FUNCTION_BLOCK SPECIALSTRING_EQ (* Basic Function Block Type *)
  (* Standard: 61499-2 *)
  (* Version 0.0, 2015-11-04, 4DIAC-IDE, 4DIAC-Consortium *)
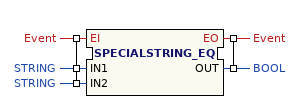
  EVENT_INPUT
    EI WITH IN1, IN2; (* Initialization Request *)
  END_EVENT
  EVENT_OUTPUT
    EO WITH OUT; (* Initialization Confirm *)
  END_EVENT
  VAR_INPUT
    IN1 : STRING;
    IN2 : STRING;
  END_VAR
  VAR_OUTPUT
    OUT : BOOL;
  END_VAR
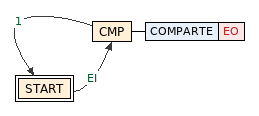
  EC_STATES
    START; (* Initial State *)
    CMP : COMPARTE -> EO; (* Initialization *)
  END_STATES
  EC_TRANSITIONS
    START TO CMP := EI;
    CMP TO START := 1;
  END_TRANSITIONS
  ALGORITHM COMPARTE IN ST: (* Initialization algorithm *)
IF IN1 = IN2 THEN
OUT:=TRUE;
END_IF;
  END_ALGORITHM
END_FUNCTION_BLOCK
